(* CODESYS project ModuNexus_RECOVERED_2026-09-28T21-24-21.project

Project tree, tasks and I/O mapping:
  Device : CODESYS Control Win V3 x64, CODESYS, version 3.5.22.20
    application Application
      libraries: Standard, 3.5.22.0 (System); CmpBitmapPool, * (System)
      task MainTask (cyclic, interval t#20ms, priority 1) calls PLC_PRG
      task VISU_TASK (cyclic, interval 100 ms, priority 31) calls VisuElems.Visu_Prg
      program PRG_CORTE [LD]
      program PRG_ENERGIA [LD]
      global variables GVL_ENERGIA
      visualisation VISU_Menu
      visualisation VISU_Nexus
      image pool ImagePool
      program PLC_PRG [LD]
      function CalcVelocidadeEsteira [ST]
    Ethernet : Ethernet, CODESYS, version 4.2.0.0
      Modbus_TCP_Client : Modbus TCP Client, CODESYS, version 4.5.1.0
          settings: AutoReconnect = TRUE
        Modbus_TCP_Server_ENERGIA : Modbus TCP Server, CODESYS, version 4.5.0.0
            settings: Unit-ID = 255; IPAddress = [192, 168, 1, 20]; RELES.Function Code = 15; RELES.Read Offset = 0; RELES.Read Length = 0; RELES.Write Offset = 16#0000; RELES.Write Length = 8; RELES.Cycle Time = 100
            output Application.GVL_ENERGIA.xRELE_1 : BOOL  // RELES.RELES.Bit0
            output Application.GVL_ENERGIA.xRELE_2 : BOOL  // RELES.RELES.Bit1
            output Application.GVL_ENERGIA.xRELE_3 : BOOL  // RELES.RELES.Bit2
            output Application.GVL_ENERGIA.xRELE_4 : BOOL  // RELES.RELES.Bit3
            output Application.GVL_ENERGIA.xRELE_5 : BOOL  // RELES.RELES.Bit4
            output Application.GVL_ENERGIA.xRELE_6 : BOOL  // RELES.RELES.Bit5
            output Application.GVL_ENERGIA.xRELE_7 : BOOL  // RELES.RELES.Bit6
            output Application.GVL_ENERGIA.xRELE_8 : BOOL  // RELES.RELES.Bit7
            unmapped channels: RELES
        Modbus_TCP_Server_1_ESTEIRA : Modbus TCP Server, CODESYS, version 4.5.0.0
            settings: Unit-ID = 255; IPAddress = [192, 168, 1, 21]; ESTEIRA.Function Code = 15; ESTEIRA.Read Offset = 0; ESTEIRA.Read Length = 0; ESTEIRA.Write Offset = 16#0000; ESTEIRA.Write Length = 2; ESTEIRA.Cycle Time = 100; VELOCIDADE.Function Code = 16; VELOCIDADE.Read Offset = 0; VELOCIDADE.Read Length = 0; VELOCIDADE.Write Offset = 16#0000; VELOCIDADE.Write Length = 1; VELOCIDADE.Cycle Time = 100
            output xLIGAR_ESTEIRA : BOOL  // ESTEIRA.ESTEIRA.Bit0
            output xDIRECAO_ESTEIRA : BOOL  // ESTEIRA.ESTEIRA.Bit1
            output Application.GVL_ENERGIA.wVELOCIDADE_ESTEIRA : WORD  // VELOCIDADE.VELOCIDADE
            unmapped channels: ESTEIRA, VELOCIDADE
        Modbus_TCP_Server_2_FLOWPACK : Modbus TCP Server, CODESYS, version 4.5.0.0
            settings: Unit-ID = 255; IPAddress = [192, 168, 1, 22]; Channel 0.Function Code = 5; Channel 0.Read Offset = 0; Channel 0.Read Length = 0; Channel 0.Write Offset = 16#0000; Channel 0.Write Length = 1; Channel 0.Cycle Time = 100
            output LED1 : BOOL  // Channel 0.Channel 0.Bit0
            unmapped channels: Channel 0
  text list GlobalTextList
*)

// Device/Application/GVL_ENERGIA
{attribute 'qualified_only'}
VAR_GLOBAL
    xRELE_1 : BOOL; (* Coil 0 - IN1 *)
    xRELE_2 : BOOL; (* Coil 1 - IN2 *)
    xRELE_3 : BOOL; (* Coil 2 - IN3 *)
    xRELE_4 : BOOL; (* Coil 3 - IN4 *)
    xRELE_5 : BOOL; (* Coil 4 - IN5 *)
    xRELE_6 : BOOL; (* Coil 5 - IN6 *)
    xRELE_7 : BOOL; (* Coil 6 - IN7 *)
    xRELE_8 : BOOL; (* Coil 7 - IN8 *)
	(* Comandos do operador *)
	(* Comandos do operador *)
	xLIGAR_RELE_1 : BOOL;
	xLIGAR_RELE_2 : BOOL;
	xLIGAR_RELE_3 : BOOL;
	xLIGAR_RELE_4 : BOOL;
	xLIGAR_RELE_5 : BOOL;
	xLIGAR_RELE_6 : BOOL;
	xLIGAR_RELE_7 : BOOL;
	xLIGAR_RELE_8 : BOOL;
	
	xLIGAR_MODULO_ENERGIA : BOOL := TRUE;
	xLIGAR_MODULO_ESTEIRA : BOOL := TRUE;
	
	xLIGAR_ESTEIRA    : BOOL;
    xDIRECAO_ESTEIRA  : BOOL;
    wVELOCIDADE_ESTEIRA : WORD := 50;
	wVEL_SETPOINT : WORD := 75;  (* velocidade desejada, muda aqui *)

	xDESLIGADO_RELE_1: BOOL ;
	xDESLIGADO_RELE_2: BOOL ;
	xDESLIGADO_RELE_3: BOOL ;
	xDESLIGADO_RELE_4: BOOL ;
	xDESLIGADO_RELE_5: BOOL ;
	xDESLIGADO_RELE_6: BOOL ;
	xDESLIGADO_RELE_7: BOOL ;
	xDESLIGADO_RELE_8: BOOL ;
	xEMERGENCIA : BOOL := FALSE;
END_VAR

// Device/Application/PLC_PRG
PROGRAM PLC_PRG
VAR
	LIGAR_MODULO_ENERGIA: BOOL := TRUE;
	xTESTE : BOOL;
END_VAR

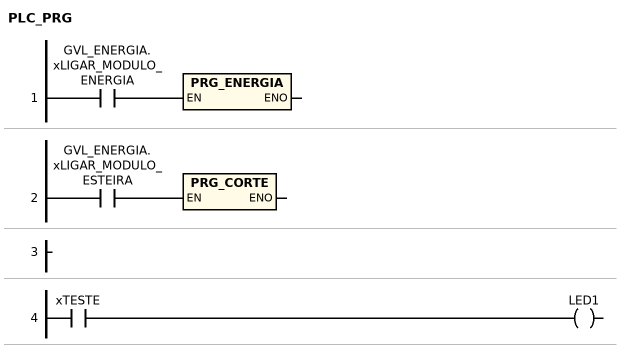
// NETWORK 1
IF GVL_ENERGIA.xLIGAR_MODULO_ENERGIA THEN PRG_ENERGIA(); END_IF

// NETWORK 2
IF GVL_ENERGIA.xLIGAR_MODULO_ESTEIRA THEN PRG_CORTE(); END_IF

// NETWORK 3

// NETWORK 4
LED1 := xTESTE;

END_PROGRAM

// Device/Application/PRG_ENERGIA
PROGRAM PRG_ENERGIA
VAR
	xEMERGENCIA : BOOL := TRUE;
	//Controle do módulo do Relé.
	//Muito importante para poder desligar módulos individualmente.
	//IMPORTANTE: RELE 4 É DO SWITCH, NORMALMENTE FECHADO, NUNCA PODE SER DESLIGADO.
	//Atenção, caso tenha o conexão com o switch interrompida, a comunicação com os módulos não terá efeito, USE OS COMANDOS FISICOS PARA DETERMINAR A PROXIMA AÇÃO.
END_VAR

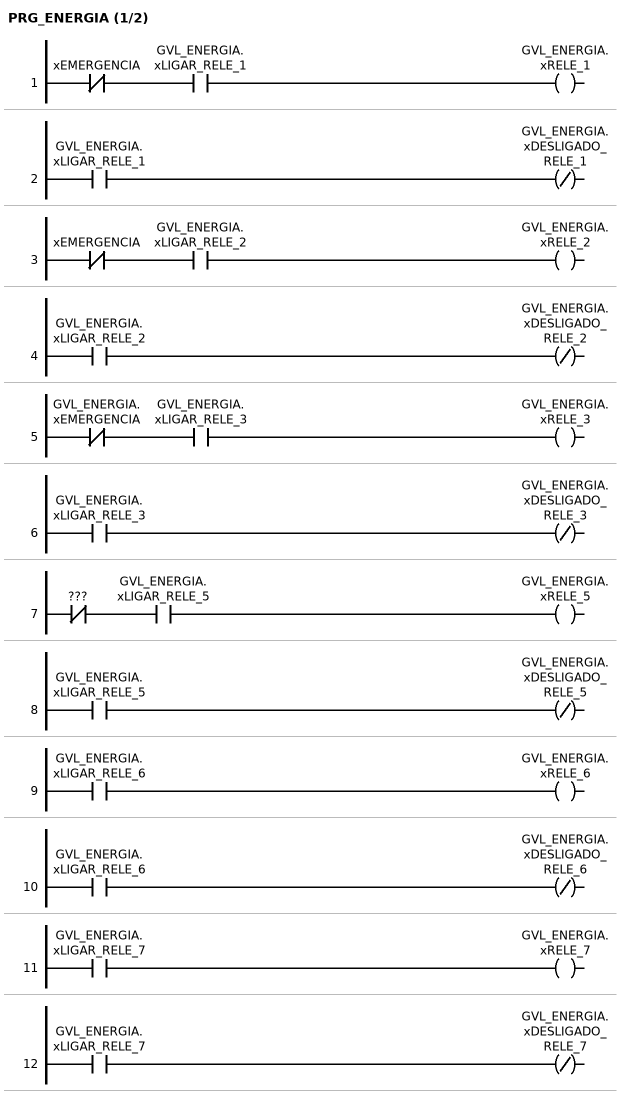
// NETWORK 1
GVL_ENERGIA.xRELE_1 := NOT xEMERGENCIA AND GVL_ENERGIA.xLIGAR_RELE_1;

// NETWORK 2
GVL_ENERGIA.xDESLIGADO_RELE_1 := NOT GVL_ENERGIA.xLIGAR_RELE_1;

// NETWORK 3
GVL_ENERGIA.xRELE_2 := NOT xEMERGENCIA AND GVL_ENERGIA.xLIGAR_RELE_2;

// NETWORK 4
GVL_ENERGIA.xDESLIGADO_RELE_2 := NOT GVL_ENERGIA.xLIGAR_RELE_2;

// NETWORK 5
GVL_ENERGIA.xRELE_3 := NOT GVL_ENERGIA.xEMERGENCIA AND GVL_ENERGIA.xLIGAR_RELE_3;

// NETWORK 6
GVL_ENERGIA.xDESLIGADO_RELE_3 := NOT GVL_ENERGIA.xLIGAR_RELE_3;

// NETWORK 7
GVL_ENERGIA.xRELE_5 := ??? AND GVL_ENERGIA.xLIGAR_RELE_5;

// NETWORK 8
GVL_ENERGIA.xDESLIGADO_RELE_5 := NOT GVL_ENERGIA.xLIGAR_RELE_5;

// NETWORK 9
GVL_ENERGIA.xRELE_6 := GVL_ENERGIA.xLIGAR_RELE_6;

// NETWORK 10
GVL_ENERGIA.xDESLIGADO_RELE_6 := NOT GVL_ENERGIA.xLIGAR_RELE_6;

// NETWORK 11
GVL_ENERGIA.xRELE_7 := GVL_ENERGIA.xLIGAR_RELE_7;

// NETWORK 12
GVL_ENERGIA.xDESLIGADO_RELE_7 := NOT GVL_ENERGIA.xLIGAR_RELE_7;

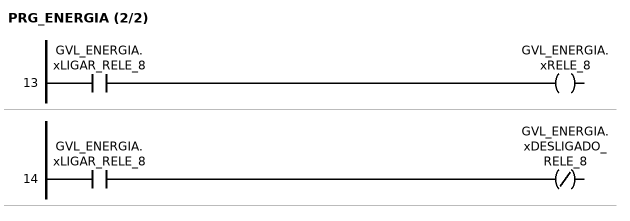
// NETWORK 13
GVL_ENERGIA.xRELE_8 := GVL_ENERGIA.xLIGAR_RELE_8;

// NETWORK 14
GVL_ENERGIA.xDESLIGADO_RELE_8 := NOT GVL_ENERGIA.xLIGAR_RELE_8;

END_PROGRAM

// Device/Application/PRG_CORTE
PROGRAM PRG_CORTE
VAR
	wVELOCIDADE : WORD := 50;
END_VAR

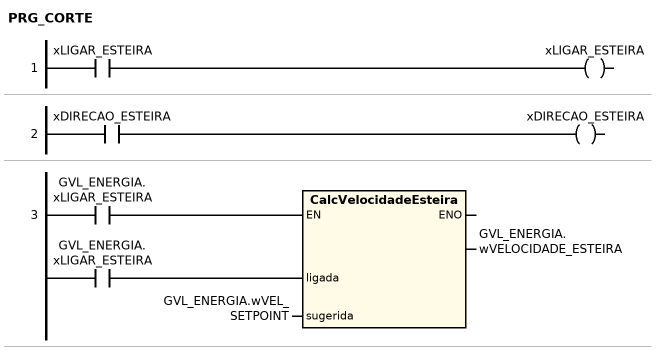
// NETWORK 1
xLIGAR_ESTEIRA := xLIGAR_ESTEIRA;

// NETWORK 2
xDIRECAO_ESTEIRA := xDIRECAO_ESTEIRA;

// NETWORK 3
IF GVL_ENERGIA.xLIGAR_ESTEIRA THEN
    GVL_ENERGIA.wVELOCIDADE_ESTEIRA := CalcVelocidadeEsteira(ligada := GVL_ENERGIA.xLIGAR_ESTEIRA, sugerida := GVL_ENERGIA.wVEL_SETPOINT);
END_IF

END_PROGRAM

// Device/Application/CalcVelocidadeEsteira
FUNCTION CalcVelocidadeEsteira : WORD
VAR_INPUT
    ligada   : BOOL;
    sugerida : WORD;
END_VAR

CalcVelocidadeEsteira := SEL(ligada, 0, LIMIT(1, sugerida, 100));

END_FUNCTION

// Device/Application/VISU_Menu
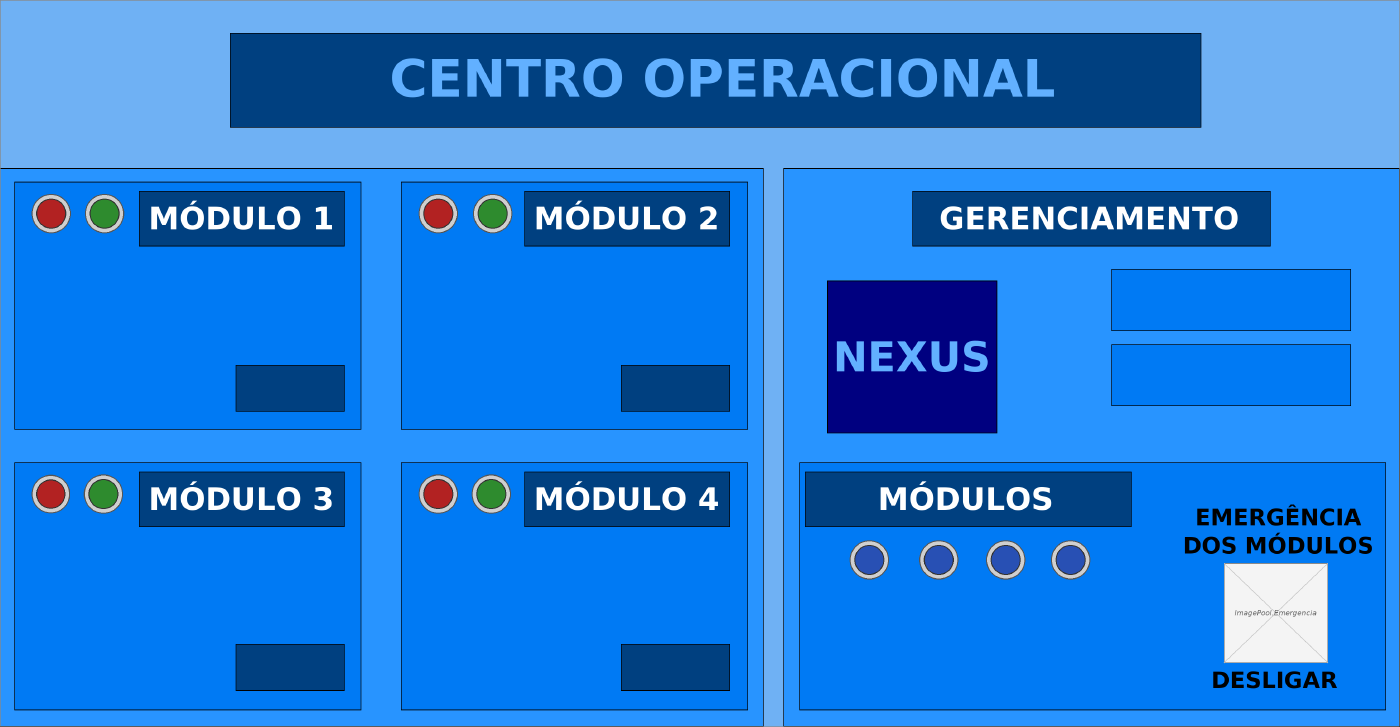
VISUALIZATION VISU_Menu  // 1955x1016
    RoundedRectangle (0,235 1066x781)
    RoundedRectangle (20,254 484x346)
    Lamp1 (113,267 66x63), variable: GVL_ENERGIA.xLIGAR_RELE_1, style: Lamp-Lamp1-Green
    Lamp1 (40,267 63x63), variable: GVL_ENERGIA.xDESLIGADO_RELE_1, style: Lamp-Lamp1-Red
    RoundedRectangle (194,267 287x77)
    Label (200,267 274x77), "MÓDULO 1"
    RoundedRectangle (560,254 484x346)
    Lamp1 (654,267 68x63), variable: GVL_ENERGIA.xLIGAR_RELE_2, style: Lamp-Lamp1-Green
    Lamp1 (580,267 64x63), variable: GVL_ENERGIA.xDESLIGADO_RELE_2, style: Lamp-Lamp1-Red
    RoundedRectangle (732,267 287x77)
    Label (738,267 274x77), "MÓDULO 2"
    RoundedRectangle (20,646 484x346)
    Lamp1 (113,659 63x63), variable: GVL_ENERGIA.xLIGAR_RELE_3, style: Lamp-Lamp1-Green
    Lamp1 (40,659 62x63), variable: GVL_ENERGIA.xDESLIGADO_RELE_3, style: Lamp-Lamp1-Red
    RoundedRectangle (194,659 287x77)
    Label (200,659 274x77), "MÓDULO 3"
    RoundedRectangle (560,646 484x346)
    Lamp1 (654,659 64x63), variable: GVL_ENERGIA.xLIGAR_RELE_5, style: Lamp-Lamp1-Green
    Lamp1 (580,659 64x63), variable: GVL_ENERGIA.xDESLIGADO_RELE_5, style: Lamp-Lamp1-Red
    RoundedRectangle (732,659 287x77)
    Label (738,659 274x77), "MÓDULO 4"
    RoundedRectangle (321,46 1356x132)
    Label (390,65 1238x89), "CENTRO OPERACIONAL"
    RoundedRectangle (1094,235 861x781)
    RoundedRectangle (1274,267 500x77)
    Label (1280,267 482x77), "GERENCIAMENTO"
    RoundedRectangle (1552,376 334x86)
    RoundedRectangle (867,900 152x65)
    RoundedRectangle (867,510 152x65)
    RoundedRectangle (329,510 152x65)
    RoundedRectangle (329,900 152x65)
    RoundedRectangle (1552,481 334x86)
    RoundedRectangle (1116,646 819x346)
    RoundedRectangle (1709,787 145x139)
        toggle PRG_ENERGIA.xEMERGENCIA
    Label (1641,681 288x123), "EMERGÊNCIA DOS MÓDULOS"
    RoundedRectangle (1124,659 456x77)
    Label (1125,659 447x77), "MÓDULOS"
    Lamp1 (1181,751 66x63), variable: GVL_ENERGIA.xLIGAR_RELE_1, style: Lamp-Lamp1-Blue
    Lamp1 (1277,751 68x63), variable: GVL_ENERGIA.xLIGAR_RELE_2, style: Lamp-Lamp1-Blue
    Lamp1 (1373,751 63x63), variable: GVL_ENERGIA.xLIGAR_RELE_3, style: Lamp-Lamp1-Blue
    Lamp1 (1463,751 64x63), variable: GVL_ENERGIA.xLIGAR_RELE_5, style: Lamp-Lamp1-Blue
    RoundedRectangle (1155,392 237x213), "NEXUS"
        OnMouseClick:  Assign=VISU_Nexus, Type=Assignment
    Image (1709,787 145x139), image: ImagePool.Emergencia
    Label (1687,928 186x45), "DESLIGAR"
END_VISUALIZATION

// Device/Application/VISU_Nexus
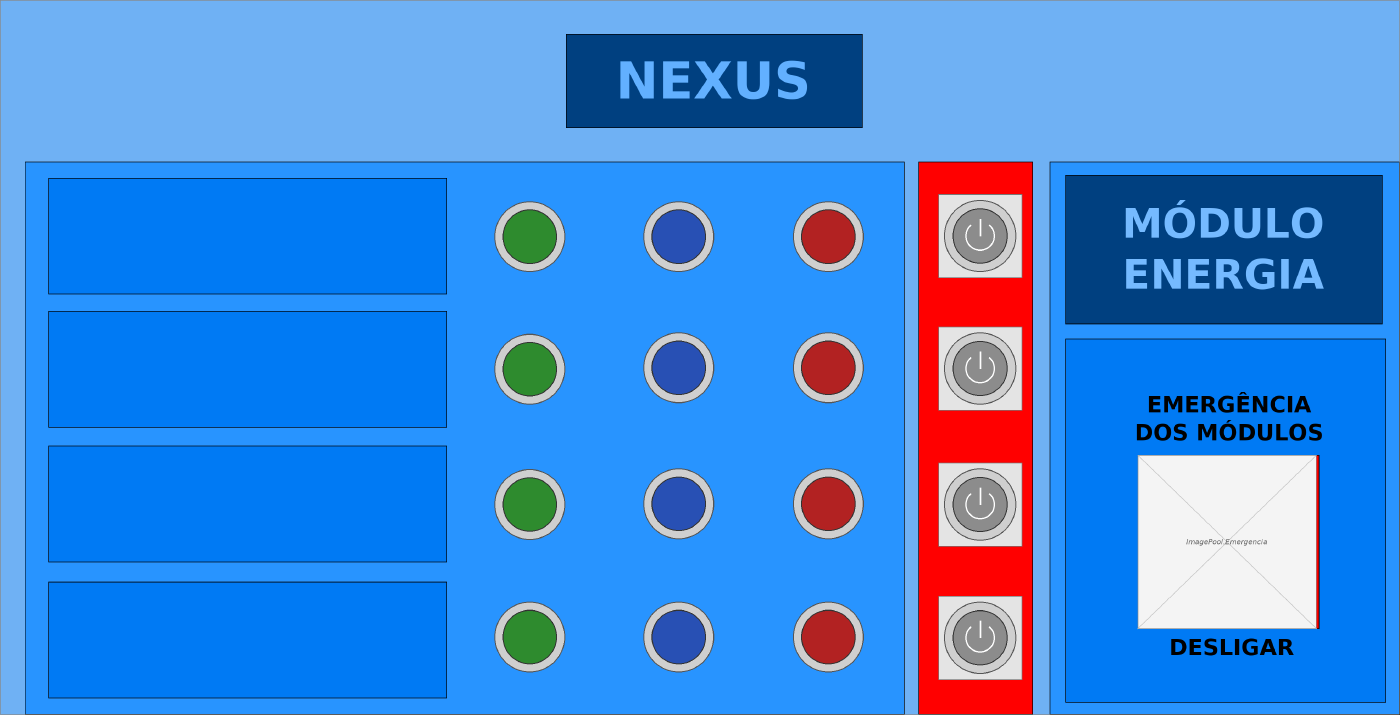
VISUALIZATION VISU_Nexus  // 1974x1009
    RoundedRectangle (35,228 1240x781)
    RoundedRectangle (798,48 418x132)
    Label (827,69 358x89), "NEXUS"
    RoundedRectangle (68,251 562x164)
    RoundedRectangle (68,439 562x164)
    RoundedRectangle (68,821 562x164)
    RoundedRectangle (68,629 562x164)
    Lamp1 (899,276 116x116), style: Lamp-Lamp1-Blue
    Lamp1 (899,461 116x116), style: Lamp-Lamp1-Blue
    Lamp1 (899,653 116x116), style: Lamp-Lamp1-Blue
    Lamp1 (899,841 116x116), style: Lamp-Lamp1-Blue
    RoundedRectangle (1295,228 161x781)
    PowerSwitch (1318,274 128x118), variable: GVL_ENERGIA.xLIGAR_RELE_1, behaviour: TOGGLE, style: Switch-PowerSwitch-Gray
    PowerSwitch (1318,461 128x118), variable: GVL_ENERGIA.xLIGAR_RELE_2, behaviour: TOGGLE, style: Switch-PowerSwitch-Gray
    PowerSwitch (1318,653 128x118), variable: GVL_ENERGIA.xLIGAR_RELE_3, behaviour: TOGGLE, style: Switch-PowerSwitch-Gray
    PowerSwitch (1318,841 128x118), variable: GVL_ENERGIA.xLIGAR_RELE_5, behaviour: TOGGLE, style: Switch-PowerSwitch-Gray
    Lamp1 (1110,276 116x116), variable: GVL_ENERGIA.xDESLIGADO_RELE_1, style: Lamp-Lamp1-Red
    Lamp1 (1110,461 116x116), variable: GVL_ENERGIA.xDESLIGADO_RELE_2, style: Lamp-Lamp1-Red
    Lamp1 (1110,653 116x116), variable: GVL_ENERGIA.xDESLIGADO_RELE_3, style: Lamp-Lamp1-Red
    Lamp1 (1110,841 116x116), variable: GVL_ENERGIA.xDESLIGADO_RELE_5, style: Lamp-Lamp1-Red
    Lamp1 (689,276 116x116), variable: GVL_ENERGIA.xLIGAR_RELE_1, style: Lamp-Lamp1-Green
    Lamp1 (689,463 116x116), variable: GVL_ENERGIA.xLIGAR_RELE_2, style: Lamp-Lamp1-Green
    Lamp1 (689,841 116x116), variable: GVL_ENERGIA.xLIGAR_RELE_5, style: Lamp-Lamp1-Green
    RoundedRectangle (1480,228 494x781)
    RoundedRectangle (1502,478 452x513)
    RoundedRectangle (1608,642 252x245)
        toggle PRG_ENERGIA.xEMERGENCIA
    Label (1589,529 288x123), "EMERGÊNCIA DOS MÓDULOS"
    Image (1604,642 252x245), image: ImagePool.Emergencia
    Label (1644,891 186x45), "DESLIGAR"
    RoundedRectangle (1502,247 447x210)
    Label (1545,247 360x208), "MÓDULO ENERGIA"
    Lamp1 (689,653 116x118), variable: GVL_ENERGIA.xLIGAR_RELE_3, style: Lamp-Lamp1-Green
END_VISUALIZATION
